# EPICS substitutions: ek9000App/Db/EL1094_mbbiDirect.substitutions
file EL1094.template
{       pattern
        {
                TERMINAL,

        }
        {
        }
}
